FUNCTION_BLOCK fileFinder (* Example for a Simple Function Block Type *)
  (* Standard: 61499-1 *)
  (* Version 1.0, 2025-07-04, user *)
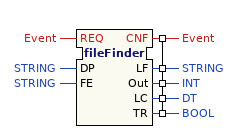
  EVENT_INPUT
    REQ; (* Normal Execution Request *)
  END_EVENT
  EVENT_OUTPUT
    CNF WITH TR, Out, LC, LF; (* Execution Confirmation *)
  END_EVENT
  VAR_INPUT
    DP : STRING;
    FE : STRING;
  END_VAR
  VAR_OUTPUT
    LF : STRING;
    Out : INT;
    LC : DT;
    TR : BOOL; (* Output *)
  END_VAR
  ALGORITHM REQ IN ST: (* Executed algorithm *)

  END_ALGORITHM
END_FUNCTION_BLOCK
